LIN {X 0,Y 92.844,Z 944.184,A -85,B 0,C 180,E1 5698.987,E2 5698.987} C_VEL
LIN {X 0,Y 90.73,Z 947.842,A -85,B 0,C 180,E1 5685.993,E2 5685.993} C_VEL
LIN {X 0,Y 91.723,Z 949.51,A -85,B 0,C 180,E1 5675.005,E2 5675.005} C_VEL
LIN {X 0,Y 92.505,Z 949.876,A -85,B 0,C 180,E1 5670.002,E2 5670.002} C_VEL
LIN {X 0,Y 91.325,Z 949.272,A -85,B 0,C 180,E1 5662.454,E2 5662.454} C_VEL
LIN {X 0,Y 90.948,Z 946.846,A -85,B 0,C 180,E1 5650.078,E2 5650.078} C_VEL
LIN {X 0,Y 94.536,Z 942.521,A -85,B 0,C 180,E1 5636.641,E2 5636.641} C_VEL
LIN {X 0,Y 102.479,Z 936.419,A -85,B 0,C 180,E1 5624.591,E2 5624.591} C_VEL
LIN {X 0,Y 114.119,Z 928.398,A -85,B 0,C 180,E1 5614.566,E2 5614.566} C_VEL
LIN {X 0,Y 127.81,Z 918.964,A -85,B 0,C 180,E1 5606.912,E2 5606.912} C_VEL
LIN {X 0,Y 143.36,Z 907.628,A -85,B 0,C 180,E1 5600.859,E2 5600.859} C_VEL
LIN {X 0,Y 158.671,Z 895.469,A -85,B 0,C 180,E1 5596.472,E2 5596.472} C_VEL
LIN {X 0,Y 174.418,Z 881.433,A -85,B 0,C 180,E1 5592.989,E2 5592.989} C_VEL
LIN {X 0,Y 189.078,Z 866.816,A -85,B 0,C 180,E1 5590.433,E2 5590.433} C_VEL
LIN {X 0,Y 203.612,Z 850.458,A -85,B 0,C 180,E1 5588.362,E2 5588.362} C_VEL
LIN {X 0,Y 216.966,Z 833.323,A -85,B 0,C 180,E1 5586.789,E2 5586.789} C_VEL
LIN {X 0,Y 229.514,Z 814.549,A -85,B 0,C 180,E1 5585.541,E2 5585.541} C_VEL
LIN {X 0,Y 240.226,Z 795.792,A -85,B 0,C 180,E1 5584.64,E2 5584.64} C_VEL
LIN {X 0,Y 250.027,Z 775.38,A -85,B 0,C 180,E1 5583.939,E2 5583.939} C_VEL
LIN {X 0,Y 258.097,Z 754.706,A -85,B 0,C 180,E1 5583.396,E2 5583.396} C_VEL
LIN {X 0,Y 264.723,Z 732.699,A -85,B 0,C 180,E1 5582.917,E2 5582.917} C_VEL
LIN {X 0,Y 269.44,Z 710.529,A -85,B 0,C 180,E1 5582.51,E2 5582.51} C_VEL
LIN {X 0,Y 273.797,Z 677.408,A -85,B 0,C 180,E1 5581.98,E2 5581.98} C_VEL
LIN {X 0,Y 280.622,Z 619.479,A -85,B 0,C 180,E1 5581.055,E2 5581.055} C_VEL
LIN {X 0,Y 280.3,Z 617.256,A -85,B 0,C 180,E1 5578.773,E2 5578.773} C_VEL
LIN {X 0,Y 280.294,Z 616.05,A -85,B 0,C 180,E1 5576.932,E2 5576.932} C_VEL
LIN {X 0,Y 280.825,Z 616.191,A -85,B 0,C 180,E1 5573.372,E2 5573.372} C_VEL
LIN {X 0,Y 271.928,Z 691.73,A -85,B 0,C 180,E1 5572.159,E2 5572.159} C_VEL
LIN {X 0,Y 268.417,Z 713.364,A -85,B 0,C 180,E1 5571.624,E2 5571.624} C_VEL
LIN {X 0,Y 263.124,Z 734.655,A -85,B 0,C 180,E1 5570.938,E2 5570.938} C_VEL
LIN {X 0,Y 256.63,Z 754.208,A -85,B 0,C 180,E1 5570.129,E2 5570.129} C_VEL
LIN {X 0,Y 248.144,Z 774.471,A -85,B 0,C 180,E1 5569.083,E2 5569.083} C_VEL
LIN {X 0,Y 238.756,Z 792.846,A -85,B 0,C 180,E1 5567.888,E2 5567.888} C_VEL
LIN {X 0,Y 227.811,Z 810.715,A -85,B 0,C 180,E1 5566.421,E2 5566.421} C_VEL
LIN {X 0,Y 215.958,Z 827.123,A -85,B 0,C 180,E1 5564.698,E2 5564.698} C_VEL
LIN {X 0,Y 203.213,Z 842.384,A -85,B 0,C 180,E1 5562.633,E2 5562.633} C_VEL
LIN {X 0,Y 190.161,Z 856.045,A -85,B 0,C 180,E1 5560.23,E2 5560.23} C_VEL
LIN {X 0,Y 175.749,Z 869.097,A -85,B 0,C 180,E1 5557.15,E2 5557.15} C_VEL
LIN {X 0,Y 161.068,Z 880.699,A -85,B 0,C 180,E1 5553.354,E2 5553.354} C_VEL
LIN {X 0,Y 145.622,Z 891.364,A -85,B 0,C 180,E1 5548.352,E2 5548.352} C_VEL
LIN {X 0,Y 131.404,Z 899.987,A -85,B 0,C 180,E1 5542.301,E2 5542.301} C_VEL
LIN {X 0,Y 118.738,Z 906.838,A -85,B 0,C 180,E1 5534.98,E2 5534.98} C_VEL
LIN {X 0,Y 107.275,Z 912.346,A -85,B 0,C 180,E1 5525.295,E2 5525.295} C_VEL
LIN {X 0,Y 99.249,Z 915.894,A -85,B 0,C 180,E1 5514.391,E2 5514.391} C_VEL
LIN {X 0,Y 94.559,Z 917.938,A -85,B 0,C 180,E1 5502.206,E2 5502.206} C_VEL
LIN {X 0,Y 93.166,Z 918.618,A -85,B 0,C 180,E1 5489.998,E2 5489.998} C_VEL
LIN {X 0,Y 94.542,Z 917.965,A -85,B 0,C 180,E1 5477.788,E2 5477.788} C_VEL
LIN {X 0,Y 99.523,Z 915.818,A -85,B 0,C 180,E1 5465.042,E2 5465.042} C_VEL
LIN {X 0,Y 107.684,Z 912.211,A -85,B 0,C 180,E1 5454.202,E2 5454.202} C_VEL
LIN {X 0,Y 118.704,Z 906.936,A -85,B 0,C 180,E1 5444.968,E2 5444.968} C_VEL
LIN {X 0,Y 132.017,Z 899.763,A -85,B 0,C 180,E1 5437.327,E2 5437.327} C_VEL
LIN {X 0,Y 146.299,Z 891.069,A -85,B 0,C 180,E1 5431.325,E2 5431.325} C_VEL
LIN {X 0,Y 161.798,Z 880.322,A -85,B 0,C 180,E1 5426.365,E2 5426.365} C_VEL
LIN {X 0,Y 176.517,Z 868.632,A -85,B 0,C 180,E1 5422.599,E2 5422.599} C_VEL
LIN {X 0,Y 190.96,Z 855.51,A -85,B 0,C 180,E1 5419.542,E2 5419.542} C_VEL
LIN {X 0,Y 204.916,Z 840.79,A -85,B 0,C 180,E1 5417.006,E2 5417.006} C_VEL
LIN {X 0,Y 217.824,Z 825.026,A -85,B 0,C 180,E1 5414.949,E2 5414.949} C_VEL
LIN {X 0,Y 230.026,Z 807.655,A -85,B 0,C 180,E1 5413.199,E2 5413.199} C_VEL
LIN {X 0,Y 240.54,Z 790.063,A -85,B 0,C 180,E1 5411.812,E2 5411.812} C_VEL
LIN {X 0,Y 249.749,Z 771.638,A -85,B 0,C 180,E1 5410.653,E2 5410.653} C_VEL
LIN {X 0,Y 257.613,Z 752.256,A -85,B 0,C 180,E1 5409.684,E2 5409.684} C_VEL
LIN {X 0,Y 264.302,Z 731.286,A -85,B 0,C 180,E1 5408.845,E2 5408.845} C_VEL
LIN {X 0,Y 269.249,Z 710.24,A -85,B 0,C 180,E1 5408.193,E2 5408.193} C_VEL
LIN {X 0,Y 272.587,Z 688.673,A -85,B 0,C 180,E1 5407.681,E2 5407.681} C_VEL
LIN {X 0,Y 281.045,Z 616.375,A -85,B 0,C 180,E1 5406.537,E2 5406.537} C_VEL
LIN {X 0,Y 280.546,Z 616.268,A -85,B 0,C 180,E1 5402.758,E2 5402.758} C_VEL
LIN {X 0,Y 280.78,Z 619.257,A -85,B 0,C 180,E1 5399.286,E2 5399.286} C_VEL
LIN {X 0,Y 280.825,Z 619.898,A -85,B 0,C 180,E1 5398.919,E2 5398.919} C_VEL
LIN {X 0,Y 270.217,Z 707.667,A -85,B 0,C 180,E1 5397.545,E2 5397.545} C_VEL
LIN {X 0,Y 265.614,Z 730.02,A -85,B 0,C 180,E1 5397.141,E2 5397.141} C_VEL
LIN {X 0,Y 259.397,Z 751.474,A -85,B 0,C 180,E1 5396.686,E2 5396.686} C_VEL
LIN {X 0,Y 251.51,Z 772.477,A -85,B 0,C 180,E1 5396.152,E2 5396.152} C_VEL
LIN {X 0,Y 242.245,Z 792.435,A -85,B 0,C 180,E1 5395.503,E2 5395.503} C_VEL
LIN {X 0,Y 231.466,Z 811.787,A -85,B 0,C 180,E1 5394.623,E2 5394.623} C_VEL
LIN {X 0,Y 219.378,Z 830.176,A -85,B 0,C 180,E1 5393.459,E2 5393.459} C_VEL
LIN {X 0,Y 205.994,Z 847.809,A -85,B 0,C 180,E1 5391.93,E2 5391.93} C_VEL
LIN {X 0,Y 201.298,Z 853.523,A -85,B 0,C 180,E1 5391.329,E2 5391.329} C_VEL
LIN {X 0,Y 196.029,Z 859.15,A -85,B 0,C 180,E1 5390.925,E2 5390.925} C_VEL
LIN {X 0,Y 181.094,Z 872.632,A -85,B 0,C 180,E1 5390.728,E2 5390.728} C_VEL
LIN {X 0,Y 175.524,Z 877.637,A -85,B 0,C 180,E1 5390.186,E2 5390.186} C_VEL
LIN {X 0,Y 159.92,Z 891.306,A -85,B 0,C 180,E1 5387.232,E2 5387.232} C_VEL
LIN {X 0,Y 143.148,Z 904.418,A -85,B 0,C 180,E1 5383.105,E2 5383.105} C_VEL
LIN {X 0,Y 127.381,Z 915.559,A -85,B 0,C 180,E1 5377.843,E2 5377.843} C_VEL
LIN {X 0,Y 112.128,Z 925.478,A -85,B 0,C 180,E1 5370.632,E2 5370.632} C_VEL
LIN {X 0,Y 98.931,Z 933.637,A -85,B 0,C 180,E1 5361.093,E2 5361.093} C_VEL
LIN {X 0,Y 89.055,Z 940.095,A -85,B 0,C 180,E1 5348.955,E2 5348.955} C_VEL
LIN {X 0,Y 83.675,Z 944.812,A -85,B 0,C 180,E1 5334.723,E2 5334.723} C_VEL
LIN {X 0,Y 82.925,Z 947.381,A -85,B 0,C 180,E1 5321.829,E2 5321.829} C_VEL
LIN {X 0,Y 84.428,Z 948.475,A -85,B 0,C 180,E1 5311.359,E2 5311.359} C_VEL
LIN {X 0,Y 84.428,Z 948.471,A -85,B 0,C 180,E1 5308.645,E2 5308.645} C_VEL
LIN {X 0,Y 82.927,Z 947.367,A -85,B 0,C 180,E1 5298.176,E2 5298.176} C_VEL
LIN {X 0,Y 83.818,Z 944.62,A -85,B 0,C 180,E1 5284.573,E2 5284.573} C_VEL
LIN {X 0,Y 89.428,Z 939.789,A -85,B 0,C 180,E1 5270.417,E2 5270.417} C_VEL
LIN {X 0,Y 100.068,Z 932.85,A -85,B 0,C 180,E1 5257.886,E2 5257.886} C_VEL
LIN {X 0,Y 113.01,Z 924.806,A -85,B 0,C 180,E1 5248.862,E2 5248.862} C_VEL
LIN {X 0,Y 128.172,Z 914.941,A -85,B 0,C 180,E1 5241.846,E2 5241.846} C_VEL
LIN {X 0,Y 144,Z 903.661,A -85,B 0,C 180,E1 5236.649,E2 5236.649} C_VEL
LIN {X 0,Y 160.848,Z 890.361,A -85,B 0,C 180,E1 5232.565,E2 5232.565} C_VEL
LIN {X 0,Y 176.453,Z 876.537,A -85,B 0,C 180,E1 5229.654,E2 5229.654} C_VEL
LIN {X 0,Y 192.028,Z 860.943,A -85,B 0,C 180,E1 5227.349,E2 5227.349} C_VEL
LIN {X 0,Y 206.435,Z 844.331,A -85,B 0,C 180,E1 5225.61,E2 5225.61} C_VEL
LIN {X 0,Y 219.56,Z 826.962,A -85,B 0,C 180,E1 5224.295,E2 5224.295} C_VEL
LIN {X 0,Y 231.817,Z 808.167,A -85,B 0,C 180,E1 5223.267,E2 5223.267} C_VEL
LIN {X 0,Y 242.175,Z 789.572,A -85,B 0,C 180,E1 5222.537,E2 5222.537} C_VEL
LIN {X 0,Y 251.583,Z 769.062,A -85,B 0,C 180,E1 5221.96,E2 5221.96} C_VEL
LIN {X 0,Y 259.271,Z 748.169,A -85,B 0,C 180,E1 5221.491,E2 5221.491} C_VEL
LIN {X 0,Y 265.605,Z 725.543,A -85,B 0,C 180,E1 5221.062,E2 5221.062} C_VEL
LIN {X 0,Y 269.904,Z 703.445,A -85,B 0,C 180,E1 5220.698,E2 5220.698} C_VEL
LIN {X 0,Y 279.38,Z 625.876,A -85,B 0,C 180,E1 5219.487,E2 5219.487} C_VEL
LIN {X 0,Y 279.32,Z 623.992,A -85,B 0,C 180,E1 5216.922,E2 5216.922} C_VEL
LIN {X 0,Y 279.483,Z 624.083,A -85,B 0,C 180,E1 5214.893,E2 5214.893} C_VEL
LIN {X 0,Y 271.253,Z 692.687,A -85,B 0,C 180,E1 5213.829,E2 5213.829} C_VEL
LIN {X 0,Y 267.629,Z 714.512,A -85,B 0,C 180,E1 5213.31,E2 5213.31} C_VEL
LIN {X 0,Y 262.212,Z 735.879,A -85,B 0,C 180,E1 5212.652,E2 5212.652} C_VEL
LIN {X 0,Y 255.502,Z 755.672,A -85,B 0,C 180,E1 5211.872,E2 5211.872} C_VEL
LIN {X 0,Y 247.045,Z 775.504,A -85,B 0,C 180,E1 5210.903,E2 5210.903} C_VEL
LIN {X 0,Y 237.698,Z 793.562,A -85,B 0,C 180,E1 5209.798,E2 5209.798} C_VEL
LIN {X 0,Y 226.554,Z 811.475,A -85,B 0,C 180,E1 5208.42,E2 5208.42} C_VEL
LIN {X 0,Y 214.435,Z 828.005,A -85,B 0,C 180,E1 5206.792,E2 5206.792} C_VEL
LIN {X 0,Y 200.999,Z 843.772,A -85,B 0,C 180,E1 5204.78,E2 5204.78} C_VEL
LIN {X 0,Y 186.752,Z 858.215,A -85,B 0,C 180,E1 5202.342,E2 5202.342} C_VEL
LIN {X 0,Y 171.976,Z 871.189,A -85,B 0,C 180,E1 5199.379,E2 5199.379} C_VEL
LIN {X 0,Y 156.85,Z 882.645,A -85,B 0,C 180,E1 5195.707,E2 5195.707} C_VEL
LIN {X 0,Y 141.621,Z 892.709,A -85,B 0,C 180,E1 5191.085,E2 5191.085} C_VEL
LIN {X 0,Y 126.705,Z 901.328,A -85,B 0,C 180,E1 5185.142,E2 5185.142} C_VEL
LIN {X 0,Y 113.288,Z 908.164,A -85,B 0,C 180,E1 5177.839,E2 5177.839} C_VEL
LIN {X 0,Y 101.402,Z 913.456,A -85,B 0,C 180,E1 5168.397,E2 5168.397} C_VEL
LIN {X 0,Y 92.429,Z 917.09,A -85,B 0,C 180,E1 5157.017,E2 5157.017} C_VEL
LIN {X 0,Y 87.019,Z 919.212,A -85,B 0,C 180,E1 5143.959,E2 5143.959} C_VEL
LIN {X 0,Y 85.286,Z 919.906,A -85,B 0,C 180,E1 5131.341,E2 5131.341} C_VEL
LIN {X 0,Y 86.527,Z 919.407,A -85,B 0,C 180,E1 5117.994,E2 5117.994} C_VEL
LIN {X 0,Y 91.097,Z 917.704,A -85,B 0,C 180,E1 5105.35,E2 5105.35} C_VEL
LIN {X 0,Y 99.877,Z 914.187,A -85,B 0,C 180,E1 5093.085,E2 5093.085} C_VEL
LIN {X 0,Y 111.373,Z 909.092,A -85,B 0,C 180,E1 5083.353,E2 5083.353} C_VEL
LIN {X 0,Y 125.225,Z 902.216,A -85,B 0,C 180,E1 5075.476,E2 5075.476} C_VEL
LIN {X 0,Y 140.01,Z 893.845,A -85,B 0,C 180,E1 5069.404,E2 5069.404} C_VEL
LIN {X 0,Y 155.15,Z 884.053,A -85,B 0,C 180,E1 5064.688,E2 5064.688} C_VEL
LIN {X 0,Y 171.061,Z 872.125,A -85,B 0,C 180,E1 5060.751,E2 5060.751} C_VEL
LIN {X 0,Y 185.813,Z 859.305,A -85,B 0,C 180,E1 5057.757,E2 5057.757} C_VEL
LIN {X 0,Y 200.048,Z 845.079,A -85,B 0,C 180,E1 5055.301,E2 5055.301} C_VEL
LIN {X 0,Y 213.551,Z 829.475,A -85,B 0,C 180,E1 5053.264,E2 5053.264} C_VEL
LIN {X 0,Y 226.049,Z 812.652,A -85,B 0,C 180,E1 5051.578,E2 5051.578} C_VEL
LIN {X 0,Y 237.105,Z 794.999,A -85,B 0,C 180,E1 5050.202,E2 5050.202} C_VEL
LIN {X 0,Y 246.538,Z 777.106,A -85,B 0,C 180,E1 5049.087,E2 5049.087} C_VEL
LIN {X 0,Y 255.063,Z 757.539,A -85,B 0,C 180,E1 5048.113,E2 5048.113} C_VEL
LIN {X 0,Y 262.097,Z 737.237,A -85,B 0,C 180,E1 5047.301,E2 5047.301} C_VEL
LIN {X 0,Y 267.563,Z 715.955,A -85,B 0,C 180,E1 5046.637,E2 5046.637} C_VEL
LIN {X 0,Y 271.206,Z 694.92,A -85,B 0,C 180,E1 5046.126,E2 5046.126} C_VEL
LIN {X 0,Y 278.084,Z 637.935,A -85,B 0,C 180,E1 5045.208,E2 5045.208} C_VEL
LIN {X 0,Y 279.749,Z 624.043,A -85,B 0,C 180,E1 5044.978,E2 5044.978} C_VEL
LIN {X 0,Y 279.553,Z 624.384,A -85,B 0,C 180,E1 5042.665,E2 5042.665} C_VEL
LIN {X 0,Y 279.599,Z 626.267,A -85,B 0,C 180,E1 5040.461,E2 5040.461} C_VEL
LIN {X 0,Y 269.68,Z 706.809,A -85,B 0,C 180,E1 5039.254,E2 5039.254} C_VEL
LIN {X 0,Y 265.028,Z 729.099,A -85,B 0,C 180,E1 5038.88,E2 5038.88} C_VEL
LIN {X 0,Y 259.031,Z 749.659,A -85,B 0,C 180,E1 5038.484,E2 5038.484} C_VEL
LIN {X 0,Y 251.095,Z 770.782,A -85,B 0,C 180,E1 5038.005,E2 5038.005} C_VEL
LIN {X 0,Y 242.183,Z 790.028,A -85,B 0,C 180,E1 5037.457,E2 5037.457} C_VEL
LIN {X 0,Y 231.334,Z 809.398,A -85,B 0,C 180,E1 5036.688,E2 5036.688} C_VEL
LIN {X 0,Y 219.569,Z 827.287,A -85,B 0,C 180,E1 5035.699,E2 5035.699} C_VEL
LIN {X 0,Y 205.961,Z 845.177,A -85,B 0,C 180,E1 5034.331,E2 5034.331} C_VEL
LIN {X 0,Y 191.561,Z 861.658,A -85,B 0,C 180,E1 5032.581,E2 5032.581} C_VEL
LIN {X 0,Y 175.524,Z 877.637,A -85,B 0,C 180,E1 5030.186,E2 5030.186} C_VEL
LIN {X 0,Y 169.809,Z 882.561,A -85,B 0,C 180,E1 5029.572,E2 5029.572} C_VEL
LIN {X 0,Y 153.411,Z 894.102,A -85,B 0,C 180,E1 5028.813,E2 5028.813} C_VEL
LIN {X 0,Y 147.382,Z 898.324,A -85,B 0,C 180,E1 5027.931,E2 5027.931} C_VEL
LIN {X 0,Y 130.392,Z 910.224,A -85,B 0,C 180,E1 5023.424,E2 5023.424} C_VEL
LIN {X 0,Y 113.052,Z 921.137,A -85,B 0,C 180,E1 5016.888,E2 5016.888} C_VEL
LIN {X 0,Y 98.404,Z 929.673,A -85,B 0,C 180,E1 5008.589,E2 5008.589} C_VEL
LIN {X 0,Y 85.461,Z 937.078,A -85,B 0,C 180,E1 4996.497,E2 4996.497} C_VEL
LIN {X 0,Y 77.368,Z 942.364,A -85,B 0,C 180,E1 4981.47,E2 4981.47} C_VEL
LIN {X 0,Y 74.887,Z 945.66,A -85,B 0,C 180,E1 4965.489,E2 4965.489} C_VEL
LIN {X 0,Y 76.112,Z 947.004,A -85,B 0,C 180,E1 4953.287,E2 4953.287} C_VEL
LIN {X 0,Y 76.575,Z 947.174,A -85,B 0,C 180,E1 4949.255,E2 4949.255} C_VEL
LIN {X 0,Y 74.968,Z 946.102,A -85,B 0,C 180,E1 4937.683,E2 4937.683} C_VEL
LIN {X 0,Y 76.2,Z 943.388,A -85,B 0,C 180,E1 4922.667,E2 4922.667} C_VEL
LIN {X 0,Y 82.69,Z 938.638,A -85,B 0,C 180,E1 4907.389,E2 4907.389} C_VEL
LIN {X 0,Y 94.483,Z 931.789,A -85,B 0,C 180,E1 4894.38,E2 4894.38} C_VEL
LIN {X 0,Y 108.421,Z 923.841,A -85,B 0,C 180,E1 4885.36,E2 4885.36} C_VEL
LIN {X 0,Y 125.27,Z 913.51,A -85,B 0,C 180,E1 4878.251,E2 4878.251} C_VEL
LIN {X 0,Y 141.816,Z 902.229,A -85,B 0,C 180,E1 4873.386,E2 4873.386} C_VEL
LIN {X 0,Y 159.197,Z 888.95,A -85,B 0,C 180,E1 4869.619,E2 4869.619} C_VEL
LIN {X 0,Y 175.989,Z 874.388,A -85,B 0,C 180,E1 4866.851,E2 4866.851} C_VEL
LIN {X 0,Y 191.626,Z 858.947,A -85,B 0,C 180,E1 4864.814,E2 4864.814} C_VEL
LIN {X 0,Y 206.282,Z 842.274,A -85,B 0,C 180,E1 4863.266,E2 4863.266} C_VEL
LIN {X 0,Y 219.097,Z 825.45,A -85,B 0,C 180,E1 4862.144,E2 4862.144} C_VEL
LIN {X 0,Y 231.55,Z 806.509,A -85,B 0,C 180,E1 4861.237,E2 4861.237} C_VEL
LIN {X 0,Y 241.951,Z 787.937,A -85,B 0,C 180,E1 4860.608,E2 4860.608} C_VEL
LIN {X 0,Y 251.436,Z 767.352,A -85,B 0,C 180,E1 4860.106,E2 4860.106} C_VEL
LIN {X 0,Y 258.937,Z 747.021,A -85,B 0,C 180,E1 4859.704,E2 4859.704} C_VEL
LIN {X 0,Y 265.295,Z 724.495,A -85,B 0,C 180,E1 4859.319,E2 4859.319} C_VEL
LIN {X 0,Y 269.63,Z 702.462,A -85,B 0,C 180,E1 4858.984,E2 4858.984} C_VEL
LIN {X 0,Y 278.304,Z 632.676,A -85,B 0,C 180,E1 4857.941,E2 4857.941} C_VEL
LIN {X 0,Y 278.362,Z 631.87,A -85,B 0,C 180,E1 4856.435,E2 4856.435} C_VEL
LIN {X 0,Y 270.676,Z 694.555,A -85,B 0,C 180,E1 4855.487,E2 4855.487} C_VEL
LIN {X 0,Y 266.991,Z 716.015,A -85,B 0,C 180,E1 4854.994,E2 4854.994} C_VEL
LIN {X 0,Y 261.447,Z 737.418,A -85,B 0,C 180,E1 4854.365,E2 4854.365} C_VEL
LIN {X 0,Y 254.513,Z 757.395,A -85,B 0,C 180,E1 4853.618,E2 4853.618} C_VEL
LIN {X 0,Y 245.926,Z 777.09,A -85,B 0,C 180,E1 4852.708,E2 4852.708} C_VEL
LIN {X 0,Y 236.432,Z 795.06,A -85,B 0,C 180,E1 4851.673,E2 4851.673} C_VEL
LIN {X 0,Y 224.804,Z 813.402,A -85,B 0,C 180,E1 4850.344,E2 4850.344} C_VEL
LIN {X 0,Y 212.479,Z 829.798,A -85,B 0,C 180,E1 4848.819,E2 4848.819} C_VEL
LIN {X 0,Y 198.631,Z 845.628,A -85,B 0,C 180,E1 4846.907,E2 4846.907} C_VEL
LIN {X 0,Y 184.509,Z 859.582,A -85,B 0,C 180,E1 4844.681,E2 4844.681} C_VEL
LIN {X 0,Y 169.352,Z 872.552,A -85,B 0,C 180,E1 4841.884,E2 4841.884} C_VEL
LIN {X 0,Y 153.761,Z 883.995,A -85,B 0,C 180,E1 4838.398,E2 4838.398} C_VEL
LIN {X 0,Y 137.961,Z 894.052,A -85,B 0,C 180,E1 4833.97,E2 4833.97} C_VEL
LIN {X 0,Y 122.342,Z 902.668,A -85,B 0,C 180,E1 4828.195,E2 4828.195} C_VEL
LIN {X 0,Y 108.118,Z 909.502,A -85,B 0,C 180,E1 4820.96,E2 4820.96} C_VEL
LIN {X 0,Y 94.768,Z 915.021,A -85,B 0,C 180,E1 4810.846,E2 4810.846} C_VEL
LIN {X 0,Y 85.065,Z 918.564,A -85,B 0,C 180,E1 4798.805,E2 4798.805} C_VEL
LIN {X 0,Y 79.181,Z 920.599,A -85,B 0,C 180,E1 4784.624,E2 4784.624} C_VEL
LIN {X 0,Y 77.39,Z 921.255,A -85,B 0,C 180,E1 4770.738,E2 4770.738} C_VEL
LIN {X 0,Y 78.984,Z 920.681,A -85,B 0,C 180,E1 4756.082,E2 4756.082} C_VEL
LIN {X 0,Y 84.664,Z 918.762,A -85,B 0,C 180,E1 4741.811,E2 4741.811} C_VEL
LIN {X 0,Y 94.186,Z 915.333,A -85,B 0,C 180,E1 4729.644,E2 4729.644} C_VEL
LIN {X 0,Y 107.396,Z 909.882,A -85,B 0,C 180,E1 4719.404,E2 4719.404} C_VEL
LIN {X 0,Y 121.535,Z 903.183,A -85,B 0,C 180,E1 4712.079,E2 4712.079} C_VEL
LIN {X 0,Y 137.903,Z 894.232,A -85,B 0,C 180,E1 4705.974,E2 4705.974} C_VEL
LIN {X 0,Y 153.706,Z 884.21,A -85,B 0,C 180,E1 4701.543,E2 4701.543} C_VEL
LIN {X 0,Y 169.301,Z 872.802,A -85,B 0,C 180,E1 4698.055,E2 4698.055} C_VEL
LIN {X 0,Y 184.46,Z 859.863,A -85,B 0,C 180,E1 4695.255,E2 4695.255} C_VEL
LIN {X 0,Y 199.028,Z 845.495,A -85,B 0,C 180,E1 4692.963,E2 4692.963} C_VEL
LIN {X 0,Y 212.904,Z 829.607,A -85,B 0,C 180,E1 4691.055,E2 4691.055} C_VEL
LIN {X 0,Y 225.072,Z 813.405,A -85,B 0,C 180,E1 4689.554,E2 4689.554} C_VEL
LIN {X 0,Y 236.4,Z 795.561,A -85,B 0,C 180,E1 4688.262,E2 4688.262} C_VEL
LIN {X 0,Y 245.898,Z 777.706,A -85,B 0,C 180,E1 4687.227,E2 4687.227} C_VEL
LIN {X 0,Y 254.52,Z 758.09,A -85,B 0,C 180,E1 4686.316,E2 4686.316} C_VEL
LIN {X 0,Y 261.576,Z 737.912,A -85,B 0,C 180,E1 4685.558,E2 4685.558} C_VEL
LIN {X 0,Y 267.119,Z 716.629,A -85,B 0,C 180,E1 4684.93,E2 4684.93} C_VEL
LIN {X 0,Y 270.817,Z 695.494,A -85,B 0,C 180,E1 4684.441,E2 4684.441} C_VEL
LIN {X 0,Y 277.897,Z 637.864,A -85,B 0,C 180,E1 4683.556,E2 4683.556} C_VEL
LIN {X 0,Y 278.604,Z 632.051,A -85,B 0,C 180,E1 4683.452,E2 4683.452} C_VEL
LIN {X 0,Y 278.51,Z 633.117,A -85,B 0,C 180,E1 4682.008,E2 4682.008} C_VEL
LIN {X 0,Y 269.414,Z 705.765,A -85,B 0,C 180,E1 4680.971,E2 4680.971} C_VEL
LIN {X 0,Y 264.705,Z 728.1,A -85,B 0,C 180,E1 4680.626,E2 4680.626} C_VEL
LIN {X 0,Y 258.443,Z 749.287,A -85,B 0,C 180,E1 4680.258,E2 4680.258} C_VEL
LIN {X 0,Y 250.444,Z 770.239,A -85,B 0,C 180,E1 4679.836,E2 4679.836} C_VEL
LIN {X 0,Y 241.46,Z 789.365,A -85,B 0,C 180,E1 4679.359,E2 4679.359} C_VEL
LIN {X 0,Y 231.005,Z 807.844,A -85,B 0,C 180,E1 4678.718,E2 4678.718} C_VEL
LIN {X 0,Y 218.827,Z 826.175,A -85,B 0,C 180,E1 4677.826,E2 4677.826} C_VEL
LIN {X 0,Y 204.818,Z 844.29,A -85,B 0,C 180,E1 4676.585,E2 4676.585} C_VEL
LIN {X 0,Y 190.179,Z 860.701,A -85,B 0,C 180,E1 4675.007,E2 4675.007} C_VEL
LIN {X 0,Y 174.3,Z 876.188,A -85,B 0,C 180,E1 4672.894,E2 4672.894} C_VEL
LIN {X 0,Y 158.118,Z 889.997,A -85,B 0,C 180,E1 4670.17,E2 4670.17} C_VEL
LIN {X 0,Y 147.382,Z 898.324,A -85,B 0,C 180,E1 4667.931,E2 4667.931} C_VEL
LIN {X 0,Y 141.288,Z 902.454,A -85,B 0,C 180,E1 4666.943,E2 4666.943} C_VEL
LIN {X 0,Y 123.913,Z 911.916,A -85,B 0,C 180,E1 4665.249,E2 4665.249} C_VEL
LIN {X 0,Y 117.673,Z 915.286,A -85,B 0,C 180,E1 4663.798,E2 4663.798} C_VEL
LIN {X 0,Y 100.325,Z 925.021,A -85,B 0,C 180,E1 4656.467,E2 4656.467} C_VEL
LIN {X 0,Y 85.309,Z 932.836,A -85,B 0,C 180,E1 4646.316,E2 4646.316} C_VEL
LIN {X 0,Y 73.922,Z 938.854,A -85,B 0,C 180,E1 4632.553,E2 4632.553} C_VEL
LIN {X 0,Y 67.76,Z 943.017,A -85,B 0,C 180,E1 4615.336,E2 4615.336} C_VEL
LIN {X 0,Y 67.484,Z 945.365,A -85,B 0,C 180,E1 4597.665,E2 4597.665} C_VEL
LIN {X 0,Y 68.733,Z 945.874,A -85,B 0,C 180,E1 4590.003,E2 4590.003} C_VEL
LIN {X 0,Y 67.017,Z 944.836,A -85,B 0,C 180,E1 4577.072,E2 4577.072} C_VEL
LIN {X 0,Y 68.684,Z 942.154,A -85,B 0,C 180,E1 4560.34,E2 4560.34} C_VEL
LIN {X 0,Y 76.223,Z 937.487,A -85,B 0,C 180,E1 4543.834,E2 4543.834} C_VEL
LIN {X 0,Y 88.609,Z 931.091,A -85,B 0,C 180,E1 4530.968,E2 4530.968} C_VEL
LIN {X 0,Y 104.271,Z 922.87,A -85,B 0,C 180,E1 4521.564,E2 4521.564} C_VEL
LIN {X 0,Y 122.003,Z 912.598,A -85,B 0,C 180,E1 4514.777,E2 4514.777} C_VEL
LIN {X 0,Y 139.18,Z 901.429,A -85,B 0,C 180,E1 4510.24,E2 4510.24} C_VEL
LIN {X 0,Y 157.055,Z 888.268,A -85,B 0,C 180,E1 4506.774,E2 4506.774} C_VEL
LIN {X 0,Y 173.457,Z 874.539,A -85,B 0,C 180,E1 4504.36,E2 4504.36} C_VEL
LIN {X 0,Y 189.628,Z 859.027,A -85,B 0,C 180,E1 4502.48,E2 4502.48} C_VEL
LIN {X 0,Y 204.126,Z 842.958,A -85,B 0,C 180,E1 4501.122,E2 4501.122} C_VEL
LIN {X 0,Y 217.944,Z 825.325,A -85,B 0,C 180,E1 4500.059,E2 4500.059} C_VEL
LIN {X 0,Y 229.958,Z 807.544,A -85,B 0,C 180,E1 4499.3,E2 4499.3} C_VEL
LIN {X 0,Y 240.496,Z 789.157,A -85,B 0,C 180,E1 4498.748,E2 4498.748} C_VEL
LIN {X 0,Y 250.044,Z 769.101,A -85,B 0,C 180,E1 4498.317,E2 4498.317} C_VEL
LIN {X 0,Y 258.351,Z 747.381,A -85,B 0,C 180,E1 4497.938,E2 4497.938} C_VEL
LIN {X 0,Y 264.671,Z 725.796,A -85,B 0,C 180,E1 4497.607,E2 4497.607} C_VEL
LIN {X 0,Y 269.251,Z 703.844,A -85,B 0,C 180,E1 4497.299,E2 4497.299} C_VEL
LIN {X 0,Y 270.489,Z 695.338,A -85,B 0,C 180,E1 4497.172,E2 4497.172} C_VEL
LIN {X 0,Y 266.749,Z 716.82,A -85,B 0,C 180,E1 4496.702,E2 4496.702} C_VEL
LIN {X 0,Y 261.129,Z 738.225,A -85,B 0,C 180,E1 4496.11,E2 4496.11} C_VEL
LIN {X 0,Y 254.246,Z 757.873,A -85,B 0,C 180,E1 4495.424,E2 4495.424} C_VEL
LIN {X 0,Y 245.537,Z 777.703,A -85,B 0,C 180,E1 4494.575,E2 4494.575} C_VEL
LIN {X 0,Y 235.904,Z 795.775,A -85,B 0,C 180,E1 4493.613,E2 4493.613} C_VEL
LIN {X 0,Y 224.404,Z 813.704,A -85,B 0,C 180,E1 4492.419,E2 4492.419} C_VEL
LIN {X 0,Y 212.28,Z 829.754,A -85,B 0,C 180,E1 4491.057,E2 4491.057} C_VEL
LIN {X 0,Y 197.913,Z 846.066,A -85,B 0,C 180,E1 4489.266,E2 4489.266} C_VEL
LIN {X 0,Y 183.505,Z 860.146,A -85,B 0,C 180,E1 4487.212,E2 4487.212} C_VEL
LIN {X 0,Y 167.062,Z 873.914,A -85,B 0,C 180,E1 4484.464,E2 4484.464} C_VEL
LIN {X 0,Y 151.024,Z 885.347,A -85,B 0,C 180,E1 4481.194,E2 4481.194} C_VEL
LIN {X 0,Y 134.669,Z 895.395,A -85,B 0,C 180,E1 4477.003,E2 4477.003} C_VEL
LIN {X 0,Y 118.35,Z 904.008,A -85,B 0,C 180,E1 4471.463,E2 4471.463} C_VEL
LIN {X 0,Y 103.3,Z 910.84,A -85,B 0,C 180,E1 4464.383,E2 4464.383} C_VEL
LIN {X 0,Y 88.917,Z 916.358,A -85,B 0,C 180,E1 4454.193,E2 4454.193} C_VEL
LIN {X 0,Y 78.213,Z 919.898,A -85,B 0,C 180,E1 4441.604,E2 4441.604} C_VEL
LIN {X 0,Y 71.562,Z 921.929,A -85,B 0,C 180,E1 4426.222,E2 4426.222} C_VEL
LIN {X 0,Y 69.502,Z 922.583,A -85,B 0,C 180,E1 4410.821,E2 4410.821} C_VEL
LIN {X 0,Y 71.338,Z 922.011,A -85,B 0,C 180,E1 4394.555,E2 4394.555} C_VEL
LIN {X 0,Y 77.769,Z 920.096,A -85,B 0,C 180,E1 4379.052,E2 4379.052} C_VEL
LIN {X 0,Y 88.288,Z 916.668,A -85,B 0,C 180,E1 4366.307,E2 4366.307} C_VEL
LIN {X 0,Y 102.538,Z 911.218,A -85,B 0,C 180,E1 4355.973,E2 4355.973} C_VEL
LIN {X 0,Y 117.511,Z 904.523,A -85,B 0,C 180,E1 4348.797,E2 4348.797} C_VEL
LIN {X 0,Y 134.618,Z 895.575,A -85,B 0,C 180,E1 4342.938,E2 4342.938} C_VEL
LIN {X 0,Y 150.977,Z 885.559,A -85,B 0,C 180,E1 4338.745,E2 4338.745} C_VEL
LIN {X 0,Y 167.018,Z 874.156,A -85,B 0,C 180,E1 4335.473,E2 4335.473} C_VEL
LIN {X 0,Y 182.54,Z 861.225,A -85,B 0,C 180,E1 4332.862,E2 4332.862} C_VEL
LIN {X 0,Y 197.408,Z 846.877,A -85,B 0,C 180,E1 4330.73,E2 4330.73} C_VEL
LIN {X 0,Y 211.534,Z 831.02,A -85,B 0,C 180,E1 4328.961,E2 4328.961} C_VEL
LIN {X 0,Y 223.9,Z 814.864,A -85,B 0,C 180,E1 4327.569,E2 4327.569} C_VEL
LIN {X 0,Y 235.774,Z 796.439,A -85,B 0,C 180,E1 4326.331,E2 4326.331} C_VEL
LIN {X 0,Y 245.517,Z 778.308,A -85,B 0,C 180,E1 4325.359,E2 4325.359} C_VEL
LIN {X 0,Y 254.229,Z 758.636,A -85,B 0,C 180,E1 4324.512,E2 4324.512} C_VEL
LIN {X 0,Y 261.329,Z 738.485,A -85,B 0,C 180,E1 4323.807,E2 4323.807} C_VEL
LIN {X 0,Y 266.968,Z 717.073,A -85,B 0,C 180,E1 4323.214,E2 4323.214} C_VEL
LIN {X 0,Y 270.381,Z 697.981,A -85,B 0,C 180,E1 4322.78,E2 4322.78} C_VEL
LIN {X 0,Y 266.344,Z 719.892,A -85,B 0,C 180,E1 4322.479,E2 4322.479} C_VEL
LIN {X 0,Y 260.626,Z 741.371,A -85,B 0,C 180,E1 4322.16,E2 4322.16} C_VEL
LIN {X 0,Y 253.068,Z 762.539,A -85,B 0,C 180,E1 4321.808,E2 4321.808} C_VEL
LIN {X 0,Y 244.019,Z 782.702,A -85,B 0,C 180,E1 4321.414,E2 4321.414} C_VEL
LIN {X 0,Y 232.974,Z 802.952,A -85,B 0,C 180,E1 4320.867,E2 4320.867} C_VEL
LIN {X 0,Y 220.951,Z 821.515,A -85,B 0,C 180,E1 4320.14,E2 4320.14} C_VEL
LIN {X 0,Y 207.794,Z 838.909,A -85,B 0,C 180,E1 4319.174,E2 4319.174} C_VEL
LIN {X 0,Y 193.091,Z 855.599,A -85,B 0,C 180,E1 4317.865,E2 4317.865} C_VEL
LIN {X 0,Y 177.283,Z 871.221,A -85,B 0,C 180,E1 4316.12,E2 4316.12} C_VEL
LIN {X 0,Y 160.892,Z 885.405,A -85,B 0,C 180,E1 4313.845,E2 4313.845} C_VEL
LIN {X 0,Y 143.623,Z 898.534,A -85,B 0,C 180,E1 4310.711,E2 4310.711} C_VEL
LIN {X 0,Y 126.447,Z 909.943,A -85,B 0,C 180,E1 4306.54,E2 4306.54} C_VEL
LIN {X 0,Y 117.673,Z 915.286,A -85,B 0,C 180,E1 4303.798,E2 4303.798} C_VEL
LIN {X 0,Y 111.445,Z 918.584,A -85,B 0,C 180,E1 4302.147,E2 4302.147} C_VEL
LIN {X 0,Y 93.751,Z 925.736,A -85,B 0,C 180,E1 4298.538,E2 4298.538} C_VEL
LIN {X 0,Y 87.675,Z 928.254,A -85,B 0,C 180,E1 4295.944,E2 4295.944} C_VEL
LIN {X 0,Y 73.005,Z 935.056,A -85,B 0,C 180,E1 4283.903,E2 4283.903} C_VEL
LIN {X 0,Y 62.499,Z 940.268,A -85,B 0,C 180,E1 4266.293,E2 4266.293} C_VEL
LIN {X 0,Y 59.054,Z 943.239,A -85,B 0,C 180,E1 4246.73,E2 4246.73} C_VEL
LIN {X 0,Y 60.552,Z 944.482,A -85,B 0,C 180,E1 4230.949,E2 4230.949} C_VEL
LIN {X 0,Y 60.554,Z 944.477,A -85,B 0,C 180,E1 4229.057,E2 4229.057} C_VEL
LIN {X 0,Y 59.074,Z 943.106,A -85,B 0,C 180,E1 4212.268,E2 4212.268} C_VEL
LIN {X 0,Y 62.905,Z 939.987,A -85,B 0,C 180,E1 4192.626,E2 4192.626} C_VEL
LIN {X 0,Y 73.609,Z 934.744,A -85,B 0,C 180,E1 4175.425,E2 4175.425} C_VEL
LIN {X 0,Y 88.384,Z 927.851,A -85,B 0,C 180,E1 4163.624,E2 4163.624} C_VEL
LIN {X 0,Y 106.165,Z 918.917,A -85,B 0,C 180,E1 4155.289,E2 4155.289} C_VEL
LIN {X 0,Y 123.817,Z 908.966,A -85,B 0,C 180,E1 4149.917,E2 4149.917} C_VEL
LIN {X 0,Y 141.791,Z 897.454,A -85,B 0,C 180,E1 4146.071,E2 4146.071} C_VEL
LIN {X 0,Y 159.745,Z 884.155,A -85,B 0,C 180,E1 4143.228,E2 4143.228} C_VEL
LIN {X 0,Y 175.997,Z 870.389,A -85,B 0,C 180,E1 4141.273,E2 4141.273} C_VEL
LIN {X 0,Y 191.952,Z 854.947,A -85,B 0,C 180,E1 4139.749,E2 4139.749} C_VEL
LIN {X 0,Y 207.008,Z 838.146,A -85,B 0,C 180,E1 4138.599,E2 4138.599} C_VEL
LIN {X 0,Y 221.118,Z 819.669,A -85,B 0,C 180,E1 4137.723,E2 4137.723} C_VEL
LIN {X 0,Y 233.236,Z 800.974,A -85,B 0,C 180,E1 4137.115,E2 4137.115} C_VEL
LIN {X 0,Y 243.845,Z 781.557,A -85,B 0,C 180,E1 4136.688,E2 4136.688} C_VEL
LIN {X 0,Y 246.875,Z 775.4,A -85,B 0,C 180,E1 4136.571,E2 4136.571} C_VEL
LIN {X 0,Y 236.621,Z 794.77,A -85,B 0,C 180,E1 4135.651,E2 4135.651} C_VEL
LIN {X 0,Y 225.44,Z 812.339,A -85,B 0,C 180,E1 4134.608,E2 4134.608} C_VEL
LIN {X 0,Y 212.398,Z 829.718,A -85,B 0,C 180,E1 4133.295,E2 4133.295} C_VEL
LIN {X 0,Y 198.981,Z 845.032,A -85,B 0,C 180,E1 4131.805,E2 4131.805} C_VEL
LIN {X 0,Y 183.803,Z 859.837,A -85,B 0,C 180,E1 4129.896,E2 4129.896} C_VEL
LIN {X 0,Y 168.51,Z 872.602,A -85,B 0,C 180,E1 4127.665,E2 4127.665} C_VEL
LIN {X 0,Y 151.374,Z 884.906,A -85,B 0,C 180,E1 4124.632,E2 4124.632} C_VEL
LIN {X 0,Y 134.399,Z 895.302,A -85,B 0,C 180,E1 4120.855,E2 4120.855} C_VEL
LIN {X 0,Y 117.262,Z 904.231,A -85,B 0,C 180,E1 4115.817,E2 4115.817} C_VEL
LIN {X 0,Y 100.407,Z 911.554,A -85,B 0,C 180,E1 4108.9,E2 4108.9} C_VEL
LIN {X 0,Y 85.36,Z 917.013,A -85,B 0,C 180,E1 4099.575,E2 4099.575} C_VEL
LIN {X 0,Y 72.545,Z 920.956,A -85,B 0,C 180,E1 4086.338,E2 4086.338} C_VEL
LIN {X 0,Y 64.525,Z 923.149,A -85,B 0,C 180,E1 4069.927,E2 4069.927} C_VEL
LIN {X 0,Y 61.652,Z 923.871,A -85,B 0,C 180,E1 4052.785,E2 4052.785} C_VEL
LIN {X 0,Y 63.332,Z 923.451,A -85,B 0,C 180,E1 4034.382,E2 4034.382} C_VEL
LIN {X 0,Y 69.758,Z 921.841,A -85,B 0,C 180,E1 4017.972,E2 4017.972} C_VEL
LIN {X 0,Y 81.468,Z 918.373,A -85,B 0,C 180,E1 4003.608,E2 4003.608} C_VEL
LIN {X 0,Y 95.839,Z 913.377,A -85,B 0,C 180,E1 3993.429,E2 3993.429} C_VEL
LIN {X 0,Y 112.461,Z 906.514,A -85,B 0,C 180,E1 3985.828,E2 3985.828} C_VEL
LIN {X 0,Y 129.122,Z 898.353,A -85,B 0,C 180,E1 3980.463,E2 3980.463} C_VEL
LIN {X 0,Y 145.918,Z 888.659,A -85,B 0,C 180,E1 3976.417,E2 3976.417} C_VEL
LIN {X 0,Y 162.309,Z 877.5,A -85,B 0,C 180,E1 3973.286,E2 3973.286} C_VEL
LIN {X 0,Y 178.125,Z 865.003,A -85,B 0,C 180,E1 3970.816,E2 3970.816} C_VEL
LIN {X 0,Y 193.24,Z 851.167,A -85,B 0,C 180,E1 3968.817,E2 3968.817} C_VEL
LIN {X 0,Y 207.57,Z 835.882,A -85,B 0,C 180,E1 3967.156,E2 3967.156} C_VEL
LIN {X 0,Y 220.579,Z 819.557,A -85,B 0,C 180,E1 3965.8,E2 3965.8} C_VEL
LIN {X 0,Y 232.709,Z 801.676,A -85,B 0,C 180,E1 3964.639,E2 3964.639} C_VEL
LIN {X 0,Y 242.953,Z 783.772,A -85,B 0,C 180,E1 3963.708,E2 3963.708} C_VEL
LIN {X 0,Y 246.376,Z 776.967,A -85,B 0,C 180,E1 3963.395,E2 3963.395} C_VEL
LIN {X 0,Y 236.272,Z 796.326,A -85,B 0,C 180,E1 3963.007,E2 3963.007} C_VEL
LIN {X 0,Y 224.656,Z 814.875,A -85,B 0,C 180,E1 3962.457,E2 3962.457} C_VEL
LIN {X 0,Y 211.041,Z 833.403,A -85,B 0,C 180,E1 3961.66,E2 3961.66} C_VEL
LIN {X 0,Y 196.968,Z 849.886,A -85,B 0,C 180,E1 3960.651,E2 3960.651} C_VEL
LIN {X 0,Y 181.515,Z 865.598,A -85,B 0,C 180,E1 3959.28,E2 3959.28} C_VEL
LIN {X 0,Y 165.125,Z 879.991,A -85,B 0,C 180,E1 3957.466,E2 3957.466} C_VEL
LIN {X 0,Y 147.546,Z 893.491,A -85,B 0,C 180,E1 3954.926,E2 3954.926} C_VEL
LIN {X 0,Y 129.421,Z 905.647,A -85,B 0,C 180,E1 3951.42,E2 3951.42} C_VEL
LIN {X 0,Y 111.086,Z 916.428,A -85,B 0,C 180,E1 3946.413,E2 3946.413} C_VEL
LIN {X 0,Y 93.151,Z 925.663,A -85,B 0,C 180,E1 3939.031,E2 3939.031} C_VEL
LIN {X 0,Y 87.675,Z 928.254,A -85,B 0,C 180,E1 3935.944,E2 3935.944} C_VEL
LIN {X 0,Y 81.76,Z 930.67,A -85,B 0,C 180,E1 3932.932,E2 3932.932} C_VEL
LIN {X 0,Y 64.352,Z 935.622,A -85,B 0,C 180,E1 3924.121,E2 3924.121} C_VEL
LIN {X 0,Y 60.182,Z 936.972,A -85,B 0,C 180,E1 3919.497,E2 3919.497} C_VEL
LIN {X 0,Y 52.151,Z 940.938,A -85,B 0,C 180,E1 3898.13,E2 3898.13} C_VEL
LIN {X 0,Y 51.693,Z 942.818,A -85,B 0,C 180,E1 3876.668,E2 3876.668} C_VEL
LIN {X 0,Y 52.693,Z 943.174,A -85,B 0,C 180,E1 3870.004,E2 3870.004} C_VEL
LIN {X 0,Y 51.209,Z 941.834,A -85,B 0,C 180,E1 3850.62,E2 3850.62} C_VEL
LIN {X 0,Y 56.005,Z 938.816,A -85,B 0,C 180,E1 3828.572,E2 3828.572} C_VEL
LIN {X 0,Y 68.372,Z 933.59,A -85,B 0,C 180,E1 3810.383,E2 3810.383} C_VEL
LIN {X 0,Y 84.512,Z 926.789,A -85,B 0,C 180,E1 3798.854,E2 3798.854} C_VEL
LIN {X 0,Y 103.855,Z 917.692,A -85,B 0,C 180,E1 3790.928,E2 3790.928} C_VEL
LIN {X 0,Y 122.645,Z 907.533,A -85,B 0,C 180,E1 3786.029,E2 3786.029} C_VEL
LIN {X 0,Y 141.116,Z 896.043,A -85,B 0,C 180,E1 3782.675,E2 3782.675} C_VEL
LIN {X 0,Y 158.96,Z 883.123,A -85,B 0,C 180,E1 3780.282,E2 3780.282} C_VEL
LIN {X 0,Y 176.01,Z 868.944,A -85,B 0,C 180,E1 3778.558,E2 3778.558} C_VEL
LIN {X 0,Y 192.168,Z 853.483,A -85,B 0,C 180,E1 3777.273,E2 3777.273} C_VEL
LIN {X 0,Y 206.867,Z 837.276,A -85,B 0,C 180,E1 3776.346,E2 3776.346} C_VEL
LIN {X 0,Y 216.329,Z 825.329,A -85,B 0,C 180,E1 3775.845,E2 3775.845} C_VEL
LIN {X 0,Y 202.86,Z 841.202,A -85,B 0,C 180,E1 3774.562,E2 3774.562} C_VEL
LIN {X 0,Y 187.387,Z 856.798,A -85,B 0,C 180,E1 3772.902,E2 3772.902} C_VEL
LIN {X 0,Y 171.599,Z 870.423,A -85,B 0,C 180,E1 3770.948,E2 3770.948} C_VEL
LIN {X 0,Y 154.698,Z 882.865,A -85,B 0,C 180,E1 3768.441,E2 3768.441} C_VEL
LIN {X 0,Y 137.162,Z 893.763,A -85,B 0,C 180,E1 3765.217,E2 3765.217} C_VEL
LIN {X 0,Y 119.488,Z 903.047,A -85,B 0,C 180,E1 3760.987,E2 3760.987} C_VEL
LIN {X 0,Y 101.471,Z 910.955,A -85,B 0,C 180,E1 3755.014,E2 3755.014} C_VEL
LIN {X 0,Y 85.582,Z 916.768,A -85,B 0,C 180,E1 3747.252,E2 3747.252} C_VEL
LIN {X 0,Y 70.416,Z 921.272,A -85,B 0,C 180,E1 3735.222,E2 3735.222} C_VEL
LIN {X 0,Y 59.641,Z 923.9,A -85,B 0,C 180,E1 3719.082,E2 3719.082} C_VEL
LIN {X 0,Y 54.163,Z 925.106,A -85,B 0,C 180,E1 3698.488,E2 3698.488} C_VEL
LIN {X 0,Y 54.41,Z 925.083,A -85,B 0,C 180,E1 3679.408,E2 3679.408} C_VEL
LIN {X 0,Y 60.021,Z 923.847,A -85,B 0,C 180,E1 3660.016,E2 3660.016} C_VEL
LIN {X 0,Y 70.997,Z 921.163,A -85,B 0,C 180,E1 3644.093,E2 3644.093} C_VEL
LIN {X 0,Y 86.296,Z 916.62,A -85,B 0,C 180,E1 3632.247,E2 3632.247} C_VEL
LIN {X 0,Y 103.099,Z 910.432,A -85,B 0,C 180,E1 3624.279,E2 3624.279} C_VEL
LIN {X 0,Y 120.334,Z 902.778,A -85,B 0,C 180,E1 3618.708,E2 3618.708} C_VEL
LIN {X 0,Y 138.356,Z 893.229,A -85,B 0,C 180,E1 3614.464,E2 3614.464} C_VEL
LIN {X 0,Y 155.041,Z 882.822,A -85,B 0,C 180,E1 3611.43,E2 3611.43} C_VEL
LIN {X 0,Y 172.044,Z 870.304,A -85,B 0,C 180,E1 3608.922,E2 3608.922} C_VEL
LIN {X 0,Y 187.366,Z 857.084,A -85,B 0,C 180,E1 3607.028,E2 3607.028} C_VEL
LIN {X 0,Y 202.844,Z 841.541,A -85,B 0,C 180,E1 3605.369,E2 3605.369} C_VEL
LIN {X 0,Y 215.906,Z 826.271,A -85,B 0,C 180,E1 3604.126,E2 3604.126} C_VEL
LIN {X 0,Y 201.8,Z 843.37,A -85,B 0,C 180,E1 3603.351,E2 3603.351} C_VEL
LIN {X 0,Y 186.105,Z 859.788,A -85,B 0,C 180,E1 3602.274,E2 3602.274} C_VEL
LIN {X 0,Y 169.982,Z 874.436,A -85,B 0,C 180,E1 3600.871,E2 3600.871} C_VEL
LIN {X 0,Y 151.997,Z 888.589,A -85,B 0,C 180,E1 3598.857,E2 3598.857} C_VEL
LIN {X 0,Y 133.291,Z 901.229,A -85,B 0,C 180,E1 3596.031,E2 3596.031} C_VEL
LIN {X 0,Y 115.036,Z 911.923,A -85,B 0,C 180,E1 3592.215,E2 3592.215} C_VEL
LIN {X 0,Y 95.735,Z 921.759,A -85,B 0,C 180,E1 3586.225,E2 3586.225} C_VEL
LIN {X 0,Y 78.019,Z 929.682,A -85,B 0,C 180,E1 3577.32,E2 3577.32} C_VEL
LIN {X 0,Y 62.586,Z 936.026,A -85,B 0,C 180,E1 3563.012,E2 3563.012} C_VEL
LIN {X 0,Y 60.182,Z 936.972,A -85,B 0,C 180,E1 3559.497,E2 3559.497} C_VEL
LIN {X 0,Y 55.763,Z 938.437,A -85,B 0,C 180,E1 3553.331,E2 3553.331} C_VEL
LIN {X 0,Y 44.066,Z 940.693,A -85,B 0,C 180,E1 3532.044,E2 3532.044} C_VEL
LIN {X 0,Y 43.234,Z 941.131,A -85,B 0,C 180,E1 3524.073,E2 3524.073} C_VEL
LIN {X 0,Y 44.632,Z 941.816,A -85,B 0,C 180,E1 3510.004,E2 3510.004} C_VEL
LIN {X 0,Y 43.621,Z 940.323,A -85,B 0,C 180,E1 3485.64,E2 3485.64} C_VEL
LIN {X 0,Y 51.06,Z 936.991,A -85,B 0,C 180,E1 3460.222,E2 3460.222} C_VEL
LIN {X 0,Y 66.077,Z 931.636,A -85,B 0,C 180,E1 3442.648,E2 3442.648} C_VEL
LIN {X 0,Y 84.364,Z 924.475,A -85,B 0,C 180,E1 3432.316,E2 3432.316} C_VEL
LIN {X 0,Y 103.547,Z 915.799,A -85,B 0,C 180,E1 3426.042,E2 3426.042} C_VEL
LIN {X 0,Y 124.024,Z 904.954,A -85,B 0,C 180,E1 3421.74,E2 3421.74} C_VEL
LIN {X 0,Y 142.983,Z 893.233,A -85,B 0,C 180,E1 3419.006,E2 3419.006} C_VEL
LIN {X 0,Y 161.167,Z 880.184,A -85,B 0,C 180,E1 3417.081,E2 3417.081} C_VEL
LIN {X 0,Y 178.453,Z 865.711,A -85,B 0,C 180,E1 3415.71,E2 3415.71} C_VEL
LIN {X 0,Y 185.6,Z 859.06,A -85,B 0,C 180,E1 3415.211,E2 3415.211} C_VEL
LIN {X 0,Y 169.076,Z 872.886,A -85,B 0,C 180,E1 3413.402,E2 3413.402} C_VEL
LIN {X 0,Y 152.734,Z 884.612,A -85,B 0,C 180,E1 3411.257,E2 3411.257} C_VEL
LIN {X 0,Y 134.74,Z 895.466,A -85,B 0,C 180,E1 3408.35,E2 3408.35} C_VEL
LIN {X 0,Y 117.115,Z 904.405,A -85,B 0,C 180,E1 3404.652,E2 3404.652} C_VEL
LIN {X 0,Y 98.381,Z 912.295,A -85,B 0,C 180,E1 3399.208,E2 3399.208} C_VEL
LIN {X 0,Y 81.559,Z 918.105,A -85,B 0,C 180,E1 3391.95,E2 3391.95} C_VEL
LIN {X 0,Y 65.073,Z 922.609,A -85,B 0,C 180,E1 3380.186,E2 3380.186} C_VEL
LIN {X 0,Y 52.863,Z 925.233,A -85,B 0,C 180,E1 3363.256,E2 3363.256} C_VEL
LIN {X 0,Y 46.372,Z 926.435,A -85,B 0,C 180,E1 3339.928,E2 3339.928} C_VEL
LIN {X 0,Y 46.507,Z 926.427,A -85,B 0,C 180,E1 3318.84,E2 3318.84} C_VEL
LIN {X 0,Y 53.309,Z 925.18,A -85,B 0,C 180,E1 3295.759,E2 3295.759} C_VEL
LIN {X 0,Y 65.723,Z 922.499,A -85,B 0,C 180,E1 3279.118,E2 3279.118} C_VEL
LIN {X 0,Y 82.332,Z 917.957,A -85,B 0,C 180,E1 3267.566,E2 3267.566} C_VEL
LIN {X 0,Y 100.097,Z 911.768,A -85,B 0,C 180,E1 3260.132,E2 3260.132} C_VEL
LIN {X 0,Y 118.027,Z 904.117,A -85,B 0,C 180,E1 3255.055,E2 3255.055} C_VEL
LIN {X 0,Y 136.592,Z 894.571,A -85,B 0,C 180,E1 3251.242,E2 3251.242} C_VEL
LIN {X 0,Y 153.668,Z 884.175,A -85,B 0,C 180,E1 3248.535,E2 3248.535} C_VEL
LIN {X 0,Y 170.996,Z 871.661,A -85,B 0,C 180,E1 3246.304,E2 3246.304} C_VEL
LIN {X 0,Y 185.258,Z 859.644,A -85,B 0,C 180,E1 3244.741,E2 3244.741} C_VEL
LIN {X 0,Y 167.264,Z 875.475,A -85,B 0,C 180,E1 3243.435,E2 3243.435} C_VEL
LIN {X 0,Y 149.032,Z 889.252,A -85,B 0,C 180,E1 3241.694,E2 3241.694} C_VEL
LIN {X 0,Y 129.984,Z 901.654,A -85,B 0,C 180,E1 3239.211,E2 3239.211} C_VEL
LIN {X 0,Y 110.304,Z 912.566,A -85,B 0,C 180,E1 3235.583,E2 3235.583} C_VEL
LIN {X 0,Y 91.286,Z 921.573,A -85,B 0,C 180,E1 3230.304,E2 3230.304} C_VEL
LIN {X 0,Y 71.78,Z 929.516,A -85,B 0,C 180,E1 3221.291,E2 3221.291} C_VEL
LIN {X 0,Y 55.897,Z 935.291,A -85,B 0,C 180,E1 3207.213,E2 3207.213} C_VEL
LIN {X 0,Y 45.409,Z 939.318,A -85,B 0,C 180,E1 3184.926,E2 3184.926} C_VEL
LIN {X 0,Y 43.234,Z 941.131,A -85,B 0,C 180,E1 3164.073,E2 3164.073} C_VEL
LIN {X 0,Y 42.51,Z 941.26,A -85,B 0,C 180,E1 3158.382,E2 3158.382} C_VEL
LIN {X 0,Y 40.025,Z 941.035,A -85,B 0,C 180,E1 3150.906,E2 3150.906} C_VEL
LIN {X 0,Y 35.376,Z 939.769,A -85,B 0,C 180,E1 3133.005,E2 3133.005} C_VEL
LIN {X 0,Y 35.352,Z 939.643,A -85,B 0,C 180,E1 3130.441,E2 3130.441} C_VEL
LIN {X 0,Y 41.821,Z 936.871,A -85,B 0,C 180,E1 3100.102,E2 3100.102} C_VEL
LIN {X 0,Y 57.379,Z 932.078,A -85,B 0,C 180,E1 3079.809,E2 3079.809} C_VEL
LIN {X 0,Y 76.33,Z 925.605,A -85,B 0,C 180,E1 3069.042,E2 3069.042} C_VEL
LIN {X 0,Y 96.095,Z 917.586,A -85,B 0,C 180,E1 3062.885,E2 3062.885} C_VEL
LIN {X 0,Y 116.053,Z 907.886,A -85,B 0,C 180,E1 3059.012,E2 3059.012} C_VEL
LIN {X 0,Y 135.218,Z 896.961,A -85,B 0,C 180,E1 3056.489,E2 3056.489} C_VEL
LIN {X 0,Y 153.607,Z 884.782,A -85,B 0,C 180,E1 3054.737,E2 3054.737} C_VEL
LIN {X 0,Y 154.998,Z 883.757,A -85,B 0,C 180,E1 3054.626,E2 3054.626} C_VEL
LIN {X 0,Y 137.211,Z 894.661,A -85,B 0,C 180,E1 3052.269,E2 3052.269} C_VEL
LIN {X 0,Y 119.071,Z 904.031,A -85,B 0,C 180,E1 3049.215,E2 3049.215} C_VEL
LIN {X 0,Y 100.422,Z 911.984,A -85,B 0,C 180,E1 3044.94,E2 3044.94} C_VEL
LIN {X 0,Y 81.592,Z 918.385,A -85,B 0,C 180,E1 3038.622,E2 3038.622} C_VEL
LIN {X 0,Y 64.138,Z 923.034,A -85,B 0,C 180,E1 3029.011,E2 3029.011} C_VEL
LIN {X 0,Y 48.724,Z 926.185,A -85,B 0,C 180,E1 3012.613,E2 3012.613} C_VEL
LIN {X 0,Y 39.748,Z 927.649,A -85,B 0,C 180,E1 2989.08,E2 2989.08} C_VEL
LIN {X 0,Y 38.193,Z 927.825,A -85,B 0,C 180,E1 2962.474,E2 2962.474} C_VEL
LIN {X 0,Y 44.368,Z 926.992,A -85,B 0,C 180,E1 2935.708,E2 2935.708} C_VEL
LIN {X 0,Y 58.048,Z 924.468,A -85,B 0,C 180,E1 2915.949,E2 2915.949} C_VEL
LIN {X 0,Y 74.708,Z 920.432,A -85,B 0,C 180,E1 2904.49,E2 2904.49} C_VEL
LIN {X 0,Y 94.01,Z 914.397,A -85,B 0,C 180,E1 2896.833,E2 2896.833} C_VEL
LIN {X 0,Y 112.461,Z 907.158,A -85,B 0,C 180,E1 2892.065,E2 2892.065} C_VEL
LIN {X 0,Y 131.432,Z 898.05,A -85,B 0,C 180,E1 2888.548,E2 2888.548} C_VEL
LIN {X 0,Y 149.775,Z 887.361,A -85,B 0,C 180,E1 2885.953,E2 2885.953} C_VEL
LIN {X 0,Y 154.637,Z 884.212,A -85,B 0,C 180,E1 2885.339,E2 2885.339} C_VEL
LIN {X 0,Y 136.242,Z 896.484,A -85,B 0,C 180,E1 2883.619,E2 2883.619} C_VEL
LIN {X 0,Y 115.992,Z 908.041,A -85,B 0,C 180,E1 2880.975,E2 2880.975} C_VEL
LIN {X 0,Y 96.102,Z 917.673,A -85,B 0,C 180,E1 2877.113,E2 2877.113} C_VEL
LIN {X 0,Y 75.961,Z 925.824,A -85,B 0,C 180,E1 2870.805,E2 2870.805} C_VEL
LIN {X 0,Y 57.385,Z 932.13,A -85,B 0,C 180,E1 2860.193,E2 2860.193} C_VEL
LIN {X 0,Y 41.731,Z 936.929,A -85,B 0,C 180,E1 2839.695,E2 2839.695} C_VEL
LIN {X 0,Y 35.32,Z 939.711,A -85,B 0,C 180,E1 2808.148,E2 2808.148} C_VEL
LIN {X 0,Y 36.536,Z 940.454,A -85,B 0,C 180,E1 2790.005,E2 2790.005} C_VEL
LIN {X 0,Y 35.352,Z 939.643,A -85,B 0,C 180,E1 2770.441,E2 2770.441} C_VEL
LIN {X 0,Y 35.543,Z 938.814,A -85,B 0,C 180,E1 2757.951,E2 2757.951} C_VEL
LIN {X 0,Y 40.502,Z 934.82,A -85,B 0,C 180,E1 2725.955,E2 2725.955} C_VEL
LIN {X 0,Y 44.543,Z 933.536,A -85,B 0,C 180,E1 2719.962,E2 2719.962} C_VEL
LIN {X 0,Y 63.471,Z 928.178,A -85,B 0,C 180,E1 2707.12,E2 2707.12} C_VEL
LIN {X 0,Y 83.978,Z 921.062,A -85,B 0,C 180,E1 2700.364,E2 2700.364} C_VEL
LIN {X 0,Y 104.166,Z 912.478,A -85,B 0,C 180,E1 2696.498,E2 2696.498} C_VEL
LIN {X 0,Y 124.378,Z 902.25,A -85,B 0,C 180,E1 2694,E2 2694} C_VEL
LIN {X 0,Y 104.37,Z 911.083,A -85,B 0,C 180,E1 2690.61,E2 2690.61} C_VEL
LIN {X 0,Y 85.5,Z 917.802,A -85,B 0,C 180,E1 2686.045,E2 2686.045} C_VEL
LIN {X 0,Y 66.489,Z 923.049,A -85,B 0,C 180,E1 2678.78,E2 2678.78} C_VEL
LIN {X 0,Y 48.944,Z 926.596,A -85,B 0,C 180,E1 2666.522,E2 2666.522} C_VEL
LIN {X 0,Y 34.887,Z 928.638,A -85,B 0,C 180,E1 2642.983,E2 2642.983} C_VEL
LIN {X 0,Y 30.054,Z 929.243,A -85,B 0,C 180,E1 2609.993,E2 2609.993} C_VEL
LIN {X 0,Y 34.871,Z 928.662,A -85,B 0,C 180,E1 2576.987,E2 2576.987} C_VEL
LIN {X 0,Y 48.628,Z 926.705,A -85,B 0,C 180,E1 2553.724,E2 2553.724} C_VEL
LIN {X 0,Y 66.469,Z 923.131,A -85,B 0,C 180,E1 2541.158,E2 2541.158} C_VEL
LIN {X 0,Y 86.412,Z 917.624,A -85,B 0,C 180,E1 2533.618,E2 2533.618} C_VEL
LIN {X 0,Y 106.271,Z 910.467,A -85,B 0,C 180,E1 2528.945,E2 2528.945} C_VEL
LIN {X 0,Y 124.025,Z 902.588,A -85,B 0,C 180,E1 2525.959,E2 2525.959} C_VEL
LIN {X 0,Y 103.12,Z 913.067,A -85,B 0,C 180,E1 2523.336,E2 2523.336} C_VEL
LIN {X 0,Y 81.993,Z 921.861,A -85,B 0,C 180,E1 2519.139,E2 2519.139} C_VEL
LIN {X 0,Y 61.587,Z 928.847,A -85,B 0,C 180,E1 2512.008,E2 2512.008} C_VEL
LIN {X 0,Y 42.218,Z 934.206,A -85,B 0,C 180,E1 2497.463,E2 2497.463} C_VEL
LIN {X 0,Y 29.317,Z 937.546,A -85,B 0,C 180,E1 2467.875,E2 2467.875} C_VEL
LIN {X 0,Y 28.406,Z 939.085,A -85,B 0,C 180,E1 2430.007,E2 2430.007} C_VEL
LIN {X 0,Y 29.694,Z 937.408,A -85,B 0,C 180,E1 2390.239,E2 2390.239} C_VEL
LIN {X 0,Y 43.822,Z 933.728,A -85,B 0,C 180,E1 2360.723,E2 2360.723} C_VEL
LIN {X 0,Y 44.543,Z 933.536,A -85,B 0,C 180,E1 2359.962,E2 2359.962} C_VEL
LIN {X 0,Y 50.061,Z 931.882,A -85,B 0,C 180,E1 2353.673,E2 2353.673} C_VEL
LIN {X 0,Y 65.037,Z 926.259,A -85,B 0,C 180,E1 2339.563,E2 2339.563} C_VEL
LIN {X 0,Y 70.85,Z 924.311,A -85,B 0,C 180,E1 2337.324,E2 2337.324} C_VEL
LIN {X 0,Y 91.561,Z 916.793,A -85,B 0,C 180,E1 2333.51,E2 2333.51} C_VEL
LIN {X 0,Y 93.207,Z 916.125,A -85,B 0,C 180,E1 2333.222,E2 2333.222} C_VEL
LIN {X 0,Y 73.43,Z 922.116,A -85,B 0,C 180,E1 2328.589,E2 2328.589} C_VEL
LIN {X 0,Y 53.081,Z 926.619,A -85,B 0,C 180,E1 2320.331,E2 2320.331} C_VEL
LIN {X 0,Y 35.477,Z 929.234,A -85,B 0,C 180,E1 2304.798,E2 2304.798} C_VEL
LIN {X 0,Y 23.39,Z 930.422,A -85,B 0,C 180,E1 2269.855,E2 2269.855} C_VEL
LIN {X 0,Y 23.719,Z 930.414,A -85,B 0,C 180,E1 2227.698,E2 2227.698} C_VEL
LIN {X 0,Y 36.224,Z 929.178,A -85,B 0,C 180,E1 2194.099,E2 2194.099} C_VEL
LIN {X 0,Y 53.962,Z 926.506,A -85,B 0,C 180,E1 2179.102,E2 2179.102} C_VEL
LIN {X 0,Y 74.368,Z 921.966,A -85,B 0,C 180,E1 2171.065,E2 2171.065} C_VEL
LIN {X 0,Y 93.051,Z 916.298,A -85,B 0,C 180,E1 2166.688,E2 2166.688} C_VEL
LIN {X 0,Y 72.083,Z 923.996,A -85,B 0,C 180,E1 2162.967,E2 2162.967} C_VEL
LIN {X 0,Y 50.052,Z 930.379,A -85,B 0,C 180,E1 2155.42,E2 2155.42} C_VEL
LIN {X 0,Y 30.276,Z 934.764,A -85,B 0,C 180,E1 2137.623,E2 2137.623} C_VEL
LIN {X 0,Y 19.55,Z 937.225,A -85,B 0,C 180,E1 2090.986,E2 2090.986} C_VEL
LIN {X 0,Y 20.227,Z 937.708,A -85,B 0,C 180,E1 2070.01,E2 2070.01} C_VEL
LIN {X 0,Y 23.897,Z 936.006,A -85,B 0,C 180,E1 2017.369,E2 2017.369} C_VEL
LIN {X 0,Y 41.872,Z 932.247,A -85,B 0,C 180,E1 1989.619,E2 1989.619} C_VEL
LIN {X 0,Y 61.982,Z 927.067,A -85,B 0,C 180,E1 1979.786,E2 1979.786} C_VEL
LIN {X 0,Y 70.85,Z 924.311,A -85,B 0,C 180,E1 1977.324,E2 1977.324} C_VEL
LIN {X 0,Y 70.827,Z 924.169,A -85,B 0,C 180,E1 1976.524,E2 1976.524} C_VEL
LIN {X 0,Y 68.242,Z 924.543,A -85,B 0,C 180,E1 1974.723,E2 1974.723} C_VEL
LIN {X 0,Y 62.466,Z 925.769,A -85,B 0,C 180,E1 1972.66,E2 1972.66} C_VEL
LIN {X 0,Y 49.189,Z 928.259,A -85,B 0,C 180,E1 1968.046,E2 1968.046} C_VEL
LIN {X 0,Y 28.991,Z 930.856,A -85,B 0,C 180,E1 1953.702,E2 1953.702} C_VEL
LIN {X 0,Y 15.388,Z 931.784,A -85,B 0,C 180,E1 1912.93,E2 1912.93} C_VEL
LIN {X 0,Y 18.37,Z 931.698,A -85,B 0,C 180,E1 1849.211,E2 1849.211} C_VEL
LIN {X 0,Y 34.228,Z 930.322,A -85,B 0,C 180,E1 1820.808,E2 1820.808} C_VEL
LIN {X 0,Y 54.784,Z 927.295,A -85,B 0,C 180,E1 1809.765,E2 1809.765} C_VEL
LIN {X 0,Y 61.39,Z 926.049,A -85,B 0,C 180,E1 1807.748,E2 1807.748} C_VEL
LIN {X 0,Y 38.999,Z 931.375,A -85,B 0,C 180,E1 1800.926,E2 1800.926} C_VEL
LIN {X 0,Y 19.135,Z 934.745,A -85,B 0,C 180,E1 1780.163,E2 1780.163} C_VEL
LIN {X 0,Y 11.997,Z 936.321,A -85,B 0,C 180,E1 1709.265,E2 1709.265} C_VEL
LIN {X 0,Y 20.827,Z 934.478,A -85,B 0,C 180,E1 1636.278,E2 1636.278} C_VEL
LIN {X 0,Y 42.02,Z 930.674,A -85,B 0,C 180,E1 1617.722,E2 1617.722} C_VEL
LIN {X 0,Y 61.55,Z 925.947,A -85,B 0,C 180,E1 1612.21,E2 1612.21} C_VEL
LIN {X 0,Y 49.189,Z 928.259,A -85,B 0,C 180,E1 1608.046,E2 1608.046} C_VEL
LIN {X 0,Y 41.716,Z 929.497,A -85,B 0,C 180,E1 1605.847,E2 1605.847} C_VEL
LIN {X 0,Y 20.707,Z 932.483,A -85,B 0,C 180,E1 1602.541,E2 1602.541} C_VEL
LIN {X 0,Y 14.383,Z 932.964,A -85,B 0,C 180,E1 1595.509,E2 1595.509} C_VEL
LIN {X 0,Y 8.044,Z 933.138,A -85,B 0,C 180,E1 1491.547,E2 1491.547} C_VEL
LIN {X 0,Y 25.492,Z 932.321,A -85,B 0,C 180,E1 1451.302,E2 1451.302} C_VEL
LIN {X 0,Y 26.901,Z 932.2,A -85,B 0,C 180,E1 1450.124,E2 1450.124} C_VEL
LIN {X 0,Y 6.334,Z 934.517,A -85,B 0,C 180,E1 1421.366,E2 1421.366} C_VEL
LIN {X 0,Y 3.832,Z 934.948,A -85,B 0,C 180,E1 1350.052,E2 1350.052} C_VEL
LIN {X 0,Y 20.15,Z 933.072,A -85,B 0,C 180,E1 1252.819,E2 1252.819} C_VEL
LIN {X 0,Y 27.166,Z 932.123,A -85,B 0,C 180,E1 1249.791,E2 1249.791} C_VEL
LIN {X 0,Y 14.383,Z 932.964,A -85,B 0,C 180,E1 1235.509,E2 1235.509} C_VEL
LIN {X 0,Y 12.752,Z 934.961,A -85,B 0,C 180,E1 1231.511,E2 1231.511} C_VEL
LIN {X 0,Y 12.752,Z 1015.5,A -85,B 0,C 180,E1 1231.511,E2 1231.511} C_VEL
LIN {X 0,Y 12.752,Z 1015.5,A -85,B 0,C 180,E1 1231.511,E2 1231.511}

QRS_NEXT_CUT()

QRS_NEXT()
QRS_HOME()

END
